(* PLC project Sem nome, Desconhecido Sem nome 1 *)
(* stored: creationDateTime 2025-02-03T21:28:09, modificationDateTime 2025-02-03T21:40:59 *)

PROGRAM program0
  VAR
    PB1 AT %IX0.0 : BOOL;
    PB2 AT %IX0.1 : BOOL;
    LED AT %QX0.0 : BOOL;
  END_VAR

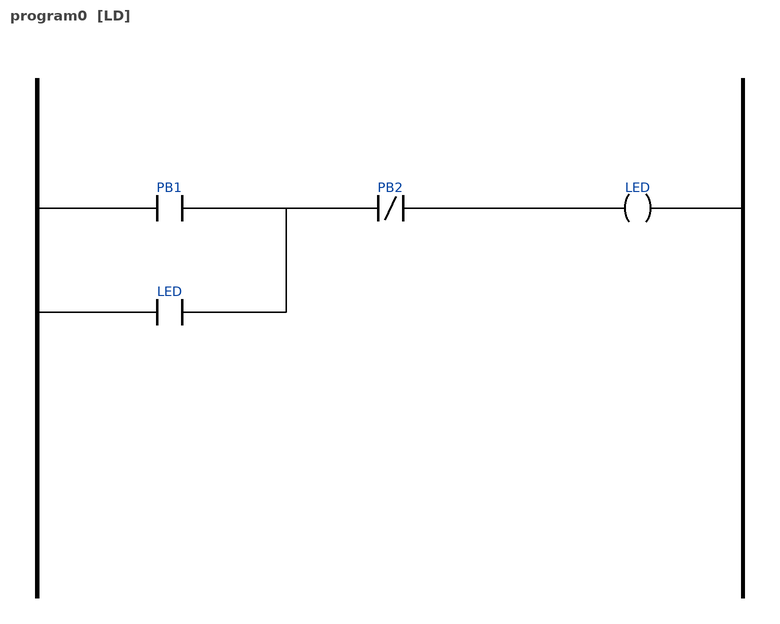
(* LD diagram, written out as Structured Text *)
LED := (PB1 OR LED) AND NOT PB2;
END_PROGRAM

CONFIGURATION Config0
  RESOURCE Res0 ON PLC
    TASK task0(INTERVAL := T#20ms, PRIORITY := 0);
    PROGRAM instance0 WITH task0 : program0;
  END_RESOURCE
END_CONFIGURATION
